             (*********************************************)
             (* parameter 3.8.3 *)
             (*********************************************)
             (
                 ParameterName_as8    := 'DOH Resistance Min',
                 ParameterType_u8     := 0,
                 attr1_u              := 0,
                 attr2_u              := 3000,
                 attr3_u              := 10,
                 UnitCode_au8         := 18,
                 Multiplier_s16       := 1,
                 Divisor_s16          := 1,
                 NumberOfDigits_u16   := 0,
                 AccesslevelCode_u8   := 179,
                 attr4_u              := 6,
                 EEPROMAddress_s      := (Page_u8 := 3, IntIndex_u8 := 186)
             ),

             (*********************************************)
             (* parameter 3.8.4 *)
             (*********************************************)
             (
                 ParameterName_as8    := 'DOH Resistance Max',
                 ParameterType_u8     := 0,
                 attr1_u              := 0,
                 attr2_u              := 3000,
                 attr3_u              := 10,
                 UnitCode_au8         := 18,
                 Multiplier_s16       := 1,
                 Divisor_s16          := 1,
                 NumberOfDigits_u16   := 0,
                 AccesslevelCode_u8   := 179,
                 attr4_u              := 44,
                 EEPROMAddress_s      := (Page_u8 := 3, IntIndex_u8 := 187)
             ),

             (*********************************************)
             (* parameter 3.8.5 *)
             (*********************************************)
             (
             ),

             (*********************************************)
             (* parameter 3.8.6 *)
             (*********************************************)
             (
             ),

             (*********************************************)
             (* parameter 3.8.7 *)
             (*********************************************)
             (
             ),

             (*********************************************)
             (* parameter 3.8.8 *)
             (*********************************************)
             (
             )

           )

           ),

      (*********************************************)
     (* parameter menu 4 - up to 8 groups can be defined here *)
     (*********************************************)
     (
         MenuName_as8    := 'Menu 4',

         ParameterGroup_as    := 

           (*********************************************)
           (* parameter group 4.1 - up to 8 parameters can be defined here *)
           (*********************************************)
           (
             (*********************************************)
             (* parameter 4.1.1 *)
             (*********************************************)
             (
             ),

             (*********************************************)
             (* parameter 4.1.2 *)
             (*********************************************)
             (
             ),

             (*********************************************)
             (* parameter 4.1.3 *)
             (*********************************************)
             (
             ),

             (*********************************************)
             (* parameter 4.1.4 *)
             (*********************************************)
             (
             ),

             (*********************************************)
             (* parameter 4.1.5 *)
             (*********************************************)
             (
             ),

             (*********************************************)
             (* parameter 4.1.6 *)
             (*********************************************)
             (
             ),

             (*********************************************)
             (* parameter 4.1.7 *)
             (*********************************************)
             (
             ),

             (*********************************************)
             (* parameter 4.1.8 *)
             (*********************************************)
             (
             )

           ),

           (*********************************************)
           (* parameter group 4.2 - up to 8 parameters can be defined here *)
           (*********************************************)
           (
             (*********************************************)
             (* parameter 4.2.1 *)
             (*********************************************)
             (
             ),

             (*********************************************)
             (* parameter 4.2.2 *)
             (*********************************************)
             (
             ),

             (*********************************************)
             (* parameter 4.2.3 *)
             (*********************************************)
             (
             ),

             (*********************************************)
             (* parameter 4.2.4 *)
             (*********************************************)
             (
             ),

             (*********************************************)
             (* parameter 4.2.5 *)
             (*********************************************)
             (
             ),

             (*********************************************)
             (* parameter 4.2.6 *)
             (*********************************************)
             (
             ),

             (*********************************************)
             (* parameter 4.2.7 *)
             (*********************************************)
             (
             ),

             (*********************************************)
             (* parameter 4.2.8 *)
             (*********************************************)
             (
             )

           ),

           (*********************************************)
           (* parameter group 4.3 - up to 8 parameters can be defined here *)
           (*********************************************)
           (
             (*********************************************)
             (* parameter 4.3.1 *)
             (*********************************************)
             (
             ),

             (*********************************************)
             (* parameter 4.3.2 *)
             (*********************************************)
             (
             ),

             (*********************************************)
             (* parameter 4.3.3 *)
             (*********************************************)
             (
             ),

             (*********************************************)
             (* parameter 4.3.4 *)
             (*********************************************)
             (
             ),

             (*********************************************)
             (* parameter 4.3.5 *)
             (*********************************************)
             (
             ),

             (*********************************************)
             (* parameter 4.3.6 *)
             (*********************************************)
             (
             ),

             (*********************************************)
             (* parameter 4.3.7 *)
             (*********************************************)
             (
             ),

             (*********************************************)
             (* parameter 4.3.8 *)
             (*********************************************)
             (
             )

           ),

           (*********************************************)
           (* parameter group 4.4 - up to 8 parameters can be defined here *)
           (*********************************************)
           (
             (*********************************************)
             (* parameter 4.4.1 *)
             (*********************************************)
             (
             ),

             (*********************************************)
             (* parameter 4.4.2 *)
             (*********************************************)
             (
             ),

             (*********************************************)
             (* parameter 4.4.3 *)
             (*********************************************)
             (
             ),

             (*********************************************)
             (* parameter 4.4.4 *)
             (*********************************************)
             (
             ),

             (*********************************************)
             (* parameter 4.4.5 *)
             (*********************************************)
             (
             ),

             (*********************************************)
             (* parameter 4.4.6 *)
             (*********************************************)
             (
             ),

             (*********************************************)
             (* parameter 4.4.7 *)
             (*********************************************)
             (
             ),

             (*********************************************)
             (* parameter 4.4.8 *)
             (*********************************************)
             (
             )

           ),

           (*********************************************)
           (* parameter group 4.5 - up to 8 parameters can be defined here *)
           (*********************************************)
           (
             (*********************************************)
             (* parameter 4.5.1 *)
             (*********************************************)
             (
             ),

             (*********************************************)
             (* parameter 4.5.2 *)
             (*********************************************)
             (
             ),

             (*********************************************)
             (* parameter 4.5.3 *)
             (*********************************************)
             (
             ),

             (*********************************************)
             (* parameter 4.5.4 *)
             (*********************************************)
             (
             ),

             (*********************************************)
             (* parameter 4.5.5 *)
             (*********************************************)
             (
             ),

             (*********************************************)
             (* parameter 4.5.6 *)
             (*********************************************)
             (
             ),

             (*********************************************)
             (* parameter 4.5.7 *)
             (*********************************************)
             (
             ),

             (*********************************************)
             (* parameter 4.5.8 *)
             (*********************************************)
             (
             )

           ),

           (*********************************************)
           (* parameter group 4.6 - up to 8 parameters can be defined here *)
           (*********************************************)
           (
             (*********************************************)
             (* parameter 4.6.1 *)
             (*********************************************)
             (
             ),

             (*********************************************)
             (* parameter 4.6.2 *)
             (*********************************************)
             (
             ),

             (*********************************************)
             (* parameter 4.6.3 *)
             (*********************************************)
             (
             ),

             (*********************************************)
             (* parameter 4.6.4 *)
             (*********************************************)
             (
             ),

             (*********************************************)
             (* parameter 4.6.5 *)
             (*********************************************)
             (
             ),

             (*********************************************)
             (* parameter 4.6.6 *)
             (*********************************************)
             (
             ),

             (*********************************************)
             (* parameter 4.6.7 *)
             (*********************************************)
             (
             ),

             (*********************************************)
             (* parameter 4.6.8 *)
             (*********************************************)
             (
             )

           ),

           (*********************************************)
           (* parameter group 4.7 - up to 8 parameters can be defined here *)
           (*********************************************)
           (
             (*********************************************)
             (* parameter 4.7.1 *)
             (*********************************************)
             (
             ),

             (*********************************************)
             (* parameter 4.7.2 *)
             (*********************************************)
             (
             ),

             (*********************************************)
             (* parameter 4.7.3 *)
             (*********************************************)
             (
             ),

             (*********************************************)
             (* parameter 4.7.4 *)
             (*********************************************)
             (
             ),

             (*********************************************)
             (* parameter 4.7.5 *)
             (*********************************************)
             (
             ),

             (*********************************************)
             (* parameter 4.7.6 *)
             (*********************************************)
             (
             ),

             (*********************************************)
             (* parameter 4.7.7 *)
             (*********************************************)
             (
             ),

             (*********************************************)
             (* parameter 4.7.8 *)
             (*********************************************)
             (
             )

           ),

           (*********************************************)
           (* parameter group 4.8 - up to 8 parameters can be defined here *)
           (*********************************************)
           (
             (*********************************************)
             (* parameter 4.8.1 *)
             (*********************************************)
             (
             ),

             (*********************************************)
             (* parameter 4.8.2 *)
             (*********************************************)
             (
             ),

             (*********************************************)
             (* parameter 4.8.3 *)
             (*********************************************)
             (
             ),

             (*********************************************)
             (* parameter 4.8.4 *)
             (*********************************************)
             (
             ),

             (*********************************************)
             (* parameter 4.8.5 *)
             (*********************************************)
             (
             ),

             (*********************************************)
             (* parameter 4.8.6 *)
             (*********************************************)
             (
             ),

             (*********************************************)
             (* parameter 4.8.7 *)
             (*********************************************)
             (
             ),

             (*********************************************)
             (* parameter 4.8.8 *)
             (*********************************************)
             (
             )

           )

           ),

      (*********************************************)
     (* parameter menu 5 - up to 8 groups can be defined here *)
     (*********************************************)
     (
         MenuName_as8    := 'Menu 5',

         ParameterGroup_as    := 

           (*********************************************)
           (* parameter group 5.1 - up to 8 parameters can be defined here *)
           (*********************************************)
           (
             (*********************************************)
             (* parameter 5.1.1 *)
             (*********************************************)
             (
             ),

             (*********************************************)
             (* parameter 5.1.2 *)
             (*********************************************)
             (
             ),

             (*********************************************)
             (* parameter 5.1.3 *)
             (*********************************************)
             (
             ),

             (*********************************************)
             (* parameter 5.1.4 *)
             (*********************************************)
             (
             ),

             (*********************************************)
             (* parameter 5.1.5 *)
             (*********************************************)
             (
             ),

             (*********************************************)
             (* parameter 5.1.6 *)
             (*********************************************)
             (
             ),

             (*********************************************)
             (* parameter 5.1.7 *)
             (*********************************************)
             (
             ),

             (*********************************************)
             (* parameter 5.1.8 *)
             (*********************************************)
             (
             )

           ),

           (*********************************************)
           (* parameter group 5.2 - up to 8 parameters can be defined here *)
           (*********************************************)
           (
             (*********************************************)
             (* parameter 5.2.1 *)
             (*********************************************)
             (
             ),

             (*********************************************)
             (* parameter 5.2.2 *)
             (*********************************************)
             (
             ),

             (*********************************************)
             (* parameter 5.2.3 *)
             (*********************************************)
             (
             ),

             (*********************************************)
             (* parameter 5.2.4 *)
             (*********************************************)
             (
             ),

             (*********************************************)
             (* parameter 5.2.5 *)
             (*********************************************)
             (
             ),

             (*********************************************)
             (* parameter 5.2.6 *)
             (*********************************************)
             (
             ),

             (*********************************************)
             (* parameter 5.2.7 *)
             (*********************************************)
             (
             ),

             (*********************************************)
             (* parameter 5.2.8 *)
             (*********************************************)
             (
             )

           ),

           (*********************************************)
           (* parameter group 5.3 - up to 8 parameters can be defined here *)
           (*********************************************)
           (
             (*********************************************)
             (* parameter 5.3.1 *)
             (*********************************************)
             (
             ),

             (*********************************************)
             (* parameter 5.3.2 *)
             (*********************************************)
             (
             ),

             (*********************************************)
             (* parameter 5.3.3 *)
             (*********************************************)
             (
             ),

             (*********************************************)
             (* parameter 5.3.4 *)
             (*********************************************)
             (
             ),

             (*********************************************)
             (* parameter 5.3.5 *)
             (*********************************************)
             (
             ),

             (*********************************************)
             (* parameter 5.3.6 *)
             (*********************************************)
             (
             ),

             (*********************************************)
             (* parameter 5.3.7 *)
             (*********************************************)
             (
             ),

             (*********************************************)
             (* parameter 5.3.8 *)
             (*********************************************)
             (
             )

           ),

           (*********************************************)
           (* parameter group 5.4 - up to 8 parameters can be defined here *)
           (*********************************************)
           (
             (*********************************************)
             (* parameter 5.4.1 *)
             (*********************************************)
             (
             ),

             (*********************************************)
             (* parameter 5.4.2 *)
             (*********************************************)
             (
             ),

             (*********************************************)
             (* parameter 5.4.3 *)
             (*********************************************)
             (
             ),

             (*********************************************)
             (* parameter 5.4.4 *)
             (*********************************************)
             (
             ),

             (*********************************************)
             (* parameter 5.4.5 *)
             (*********************************************)
             (
             ),

             (*********************************************)
             (* parameter 5.4.6 *)
             (*********************************************)
             (
             ),

             (*********************************************)
             (* parameter 5.4.7 *)
             (*********************************************)
             (
             ),

             (*********************************************)
             (* parameter 5.4.8 *)
             (*********************************************)
             (
             )

           ),

           (*********************************************)
           (* parameter group 5.5 - up to 8 parameters can be defined here *)
           (*********************************************)
           (
             (*********************************************)
             (* parameter 5.5.1 *)
             (*********************************************)
             (
             ),

             (*********************************************)
             (* parameter 5.5.2 *)
             (*********************************************)
             (
             ),

             (*********************************************)
             (* parameter 5.5.3 *)
             (*********************************************)
             (
             ),

             (*********************************************)
             (* parameter 5.5.4 *)
             (*********************************************)
             (
             ),

             (*********************************************)
             (* parameter 5.5.5 *)
             (*********************************************)
             (
             ),

             (*********************************************)
             (* parameter 5.5.6 *)
             (*********************************************)
             (
             ),

             (*********************************************)
             (* parameter 5.5.7 *)
             (*********************************************)
             (
             ),

             (*********************************************)
             (* parameter 5.5.8 *)
             (*********************************************)
             (
             )

           ),

           (*********************************************)
           (* parameter group 5.6 - up to 8 parameters can be defined here *)
           (*********************************************)
           (
             (*********************************************)
             (* parameter 5.6.1 *)
             (*********************************************)
             (
             ),

             (*********************************************)
             (* parameter 5.6.2 *)
             (*********************************************)
             (
             ),

             (*********************************************)
             (* parameter 5.6.3 *)
             (*********************************************)
             (
             ),

             (*********************************************)
             (* parameter 5.6.4 *)
             (*********************************************)
             (
             ),

             (*********************************************)
             (* parameter 5.6.5 *)
             (*********************************************)
             (
             ),

             (*********************************************)
             (* parameter 5.6.6 *)
             (*********************************************)
             (
             ),

             (*********************************************)
             (* parameter 5.6.7 *)
             (*********************************************)
             (
             ),

             (*********************************************)
             (* parameter 5.6.8 *)
             (*********************************************)
             (
             )

           ),

           (*********************************************)
           (* parameter group 5.7 - up to 8 parameters can be defined here *)
           (*********************************************)
           (
             (*********************************************)
             (* parameter 5.7.1 *)
             (*********************************************)
             (
             ),

             (*********************************************)
             (* parameter 5.7.2 *)
             (*********************************************)
             (
             ),

             (*********************************************)
             (* parameter 5.7.3 *)
             (*********************************************)
             (
             ),

             (*********************************************)
             (* parameter 5.7.4 *)
             (*********************************************)
             (
             ),

             (*********************************************)
             (* parameter 5.7.5 *)
             (*********************************************)
             (
             ),

             (*********************************************)
             (* parameter 5.7.6 *)
             (*********************************************)
             (
             ),

             (*********************************************)
             (* parameter 5.7.7 *)
             (*********************************************)
             (
             ),

             (*********************************************)
             (* parameter 5.7.8 *)
             (*********************************************)
             (
             )

           ),

           (*********************************************)
           (* parameter group 5.8 - up to 8 parameters can be defined here *)
           (*********************************************)
           (
             (*********************************************)
             (* parameter 5.8.1 *)
             (*********************************************)
             (
             ),

             (*********************************************)
             (* parameter 5.8.2 *)
             (*********************************************)
             (
             ),

             (*********************************************)
             (* parameter 5.8.3 *)
             (*********************************************)
             (
             ),

             (*********************************************)
             (* parameter 5.8.4 *)
             (*********************************************)
             (
             ),

             (*********************************************)
             (* parameter 5.8.5 *)
             (*********************************************)
             (
             ),

             (*********************************************)
             (* parameter 5.8.6 *)
             (*********************************************)
             (
             ),

             (*********************************************)
             (* parameter 5.8.7 *)
             (*********************************************)
             (
             ),

             (*********************************************)
             (* parameter 5.8.8 *)
             (*********************************************)
             (
             )

           )

           );


*)
END_VAR
(*********************************************)
(*  DON'T MAKE ANY CHANGES TO THIS PROGRAM!! *)
(*     FILE WAS AUTOMATICALLY GENERATED!!    *)
(*********************************************)

;
END_PROGRAM
